(* IEC 61131-3 sources: SRCI/RobotLibrary/RobotLibrary/POUs/Calculation/MC_CalculateFrame, 1 file *)

(* ---- MC_CalculateFrameFB.st ---- *)
/// Calculate frame with three-point method
FUNCTION_BLOCK MC_CalculateFrameFB EXTENDS RobotLibraryBaseExecuteFB
// -------------------------------------------------------------------------
//  SRCI Robot Library
// -------------------------------------------------------------------------
//
//  Object:      CalculateFrameFB
//  Author:      Thorsten Brach
//  Date:        2024-06-09
//
//  Description:
//
//
//  Copyright:
//    (C) 2024 Thorsten Brach. All rights reserved
//             Licensed under the LGPL-3.0 license.
//
//  Disclaimer:
//    This project is provided without any guarantee and can be used for
//    private and commercial purposes. Any use is at the user’s
//    own risk and responsibility.
//
// -------------------------------------------------------------------------
VAR_INPUT
  /// command parameter
  ParCmd          : CalculateFrameParCmd;
END_VAR
VAR_OUTPUT
  /// Command is transferred and confirmed by the RC
  CommandBuffered : BOOL;
  /// Command output
  OutCmd          : CalculateFrameOutCmd;
END_VAR

VAR
  /// internal copy of command parameter
 _parCmd          : CalculateFrameParCmd;
  /// command data to send
 _command         : CalculateFrameSendData;
  /// response data received
 _response        : CalculateFrameRecvData;
  /// Incremented with each position of the input parameter "PositionsArray" sent from the PLC to the RC.
  /// Default: 0
 _dataIndex       : USINT;
  /// Set TRUE by the client, when according to the user selected "Mode" the final position of the input parameter "PositionsArray" is sent to the RC.
  /// Default: FALSE
 _dataComplete    : BOOL;
END_VAR

  SUPER^(AxesGroup := AxesGroup);

END_FUNCTION_BLOCK

METHOD CheckParameterChanged : BOOL
VAR_IN_OUT
  /// Robot assignment of function
  AxesGroup    : AxesGroup;
END_VAR

  // Check ParCmd Size is > 0, becaue MemCmp does not work correctly with size = 0
  IF (SIZEOF(ParCmd) = 0)
  THEN
    RETURN;
  END_IF

  // compare memory
  CheckParameterChanged := ( MemCmp(ADR(ParCmd), ADR(_parCmd), SIZEOF(ParCmd)) <> RobotLibraryConstants.OK );

  IF ( CheckParameterChanged )
  THEN
    // update internal copy of parameters
   _parCmd := ParCmd;
    // inc parameter sequence
   _command.ParSeq := _command.ParSeq + 1;
    // update command data
    CommandData := CreateCommandPayload(); // ( Access via reference to rCommandFB in ACR )
    // notify active command register
    AxesGroup.Acyclic.ActiveCommandRegister.NotifyParameterChanged := _uniqueID;
  END_IF

END_METHOD

METHOD INTERNAL CreateCommandPayload : SendData
// Table 6-656: Sent CMD payload (PLC to RC) of "CalculateFrame"
// --------------------------
// Header
// --------------------------
// Byte 00 : UINT       - Type HB
// Byte 01 :            - Type LB
// Byte 02 : USINT      - Reserve | ExecutionMode
// Byte 03 : USINT      - ParSeq  | Priority
// --------------------------
// Datablock
// --------------------------
// Byte 04 : USIN       - DataIndex
// Byte 05 : BOOL       - DataComplete
// Byte 06 : BYTE       - Reserve
// Byte 07 : USINT      - FrameNo
// Byte 08 : USINT      - ReferenceFrame
// Byte 09 : SINT       - Mode
// Byte 10 : REAL       - Position X  HW HB
// Byte 11 :            - Position X  HW LB
// Byte 12 :            - Position X  LW HB
// Byte 13 :            - Position X  LW LB
// Byte 14 : REAL       - Position Y  HW HB
// Byte 15 :            - Position Y  HW LB
// Byte 16 :            - Position Y  LW HB
// Byte 17 :            - Position Y  LW LB
// Byte 18 : REAL       - Position Z  HW HB
// Byte 19 :            - Position Z  HW LB
// Byte 20 :            - Position Z  LW HB
// Byte 21 :            - Position Z  LW LB
// Byte 22 : REAL       - Position Rx HW HB
// Byte 23 :            - Position Rx HW LB
// Byte 24 :            - Position Rx LW HB
// Byte 25 :            - Position Rx LW LB
// Byte 26 : REAL       - Position Ry HW HB
// Byte 27 :            - Position Ry HW LB
// Byte 28 :            - Position Ry LW HB
// Byte 29 :            - Position Ry LW LB
// Byte 30 : REAL       - Position Rz HW HB
// Byte 31 :            - Position Rz HW LB
// Byte 32 :            - Position Rz LW HB
// Byte 33 :            - Position Rz LW LB
// Byte 34 : Config     - ArmConfig   LW HB
// Byte 35 :            - ArmConfig   LW LB
// Byte 36 : TurnNumber - J1 + J2     LW HB
// Byte 37 :            - J3 + J4     LW LB
// Byte 38 :            - J5 + J6     LW LB
// Byte 39 :            - E1          LW LB
// Byte 40 : REAL       - Position E1 HW HB
// Byte 41 :            - Position E1 HW LB
// Byte 42 :            - Position E1 LW HB
// Byte 43 :            - Position E1 LW LB
// Byte 44 : REAL       - Position E2 HW HB
// Byte 45 :            - Position E2 HW LB
// Byte 46 :            - Position E2 LW HB
// Byte 47 :            - Position E2 LW LB
// Byte 48 : REAL       - Position E3 HW HB
// Byte 49 :            - Position E3 HW LB
// Byte 50 :            - Position E3 LW HB
// Byte 51 :            - Position E3 LW LB
// Byte 52 : REAL       - Position E4 HW HB
// Byte 53 :            - Position E4 HW LB
// Byte 54 :            - Position E4 LW HB
// Byte 55 :            - Position E4 LW LB
// Byte 56 : REAL       - Position E5 HW HB
// Byte 57 :            - Position E5 HW LB
// Byte 58 :            - Position E5 LW HB
// Byte 59 :            - Position E5 LW LB
// Byte 60 : REAL       - Position E6 HW HB
// Byte 61 :            - Position E6 HW LB
// Byte 62 :            - Position E6 LW HB
// Byte 63 :            - Position E6 LW LB
// --------------------------

  // set command parameter
  _command.CmdTyp         :=  CmdType.CalculateFrame;
  _command.ExecMode       :=  ExecMode;
  _command.ParSeq         := _command.ParSeq;
  _command.Priority       :=  Priority;
  _command.FrameNo        := _parCmd.FrameNo;
  _command.DataIndex      := _dataIndex;
  _command.DataComplete.0 := _dataComplete;
  _command.Reserve        := 0;
  _command.FrameNo        := _parCmd.FrameNo;
  _command.ReferenceFrame := _parCmd.ReferenceFrame;
  _command.Mode           := _parCmd.Mode;

  CASE _parCmd.Mode OF

    FrameCalculationMode.THREE_POINT_METHOD :

      CASE _dataIndex OF

        1: _command.Position := _parCmd.Origin;
        2: _command.Position := _parCmd.Position_X;
        3: _command.Position := _parCmd.Position_XY;

      END_CASE

    FrameCalculationMode.FOUR_POINT_METHOD  :

      CASE _dataIndex OF

        1: _command.Position := _parCmd.Origin;
        2: _command.Position := _parCmd.Position_X;
        3: _command.Position := _parCmd.Position_XY;
        4: _command.Position := _parCmd.OriginShift;

      END_CASE

    FrameCalculationMode.ONE_POINT_METHOD   :

     _command.Position := _parCmd.Origin;

  END_CASE

  // copy command data to header
  _cmdHeader := _command;
  // call base implementation to copy header to payload buffer
  CreateCommandPayload := SUPER^.CreateCommandPayload();

  // add command.DataIndex
  CreateCommandPayload.AddUsint(_command.DataIndex);
  // add command.DataComplete
  CreateCommandPayload.AddByte(_command.DataComplete);
  // add command.Reserve
  CreateCommandPayload.AddByte(_command.Reserve);
  // add command.FrameNo
  CreateCommandPayload.AddUsint(_command.FrameNo);
  // add command.ReferenceFrame
  CreateCommandPayload.AddUsint(_command.ReferenceFrame);
  // add command.Mode
  CreateCommandPayload.AddSint(_command.Mode);
  // add command.Position.X
  CreateCommandPayload.AddReal(_command.Position.X);
  // add command.Position.Y
  CreateCommandPayload.AddReal(_command.Position.Y);
  // add command.Position.Z
  CreateCommandPayload.AddReal(_command.Position.Z);
  // add command.Position.Rx
  CreateCommandPayload.AddReal(_command.Position.Rx);
  // add command.Position.Ry
  CreateCommandPayload.AddReal(_command.Position.Ry);
  // add command.Position.Rz
  CreateCommandPayload.AddReal(_command.Position.Rz);
  // add command.Position.Config
  CreateCommandPayload.AddArmConfig(_command.Position.Config);
  // add command.Position.TurnNumber
  CreateCommandPayload.AddTurnNumber(_command.Position.TurnNumber);
  // add command.Position.E1
  CreateCommandPayload.AddReal(_command.Position.E1);
  // add command.Position.E2
  CreateCommandPayload.AddReal(_command.Position.E2);
  // add command.Position.E3
  CreateCommandPayload.AddReal(_command.Position.E3);
  // add command.Position.E4
  CreateCommandPayload.AddReal(_command.Position.E4);
  // add command.Position.E5
  CreateCommandPayload.AddReal(_command.Position.E5);
  // add command.Position.E6
  CreateCommandPayload.AddReal(_command.Position.E6);

END_METHOD

METHOD FB_init : BOOL
VAR_INPUT
  /// if TRUE, the retain variables are initialized (warm start / cold start)
	bInitRetains : BOOL;
  /// if TRUE, the instance afterwards gets moved into the copy code (online change)
	bInCopyCode  : BOOL;
END_VAR

  MyType := 'MC_CalculateFrameFB';

  ExecMode := ExecutionMode.PARALLEL;

END_METHOD

METHOD PROTECTED OnCall
VAR_IN_OUT
  /// Robot assignment of function
  AxesGroup : AxesGroup;
END_VAR

  // call base implementation
  SUPER^.OnCall(AxesGroup := AxesGroup);

  CASE _stepCmd OF

    00:  IF ( _execute_R.Q )
         THEN
           // set busy flag
           Busy := TRUE;
           // Reset command outputs
           MemSet(ADR(OutCmd),0,SIZEOF(OutCmd));
           // apply command parameter
          _parCmd := ParCmd;
           // init parameter sequence
          _command.ParSeq := 1;
           // set timeout
           SetTimeout(PT := _timeoutCmd, rTimer := _timerCmd);
           // inc step counter
          _stepCmd := _stepCmd + 1;
  	     END_IF

    01: // inc data index
       _dataIndex := _dataIndex + 1;

        CASE _parCmd.Mode OF
          FrameCalculationMode.ONE_POINT_METHOD   :
            _dataComplete := _dataIndex >= 1;
          FrameCalculationMode.THREE_POINT_METHOD :
            _dataComplete := _dataIndex >= 3;
          FrameCalculationMode.FOUR_POINT_METHOD  :
            _dataComplete := _dataIndex >= 4;
  	    END_CASE

         // create command data
         CommandData := CreateCommandPayload();
         // Add command to active command register
        _uniqueID := AxesGroup.Acyclic.ActiveCommandRegister.AddCmd( pCommandFB := ADR(THIS^ ));
         // set timeout
         SetTimeout(PT := _timeoutCmd, rTimer := _timerCmd);
         // inc step counter
        _stepCmd := _stepCmd + 1;

    02:  // Wait for responce received
         IF ( _responseReceived )
         THEN
           // reset response received flag
          _responseReceived := FALSE;

           CASE  _response.State
           OF
             CmdMessageState.BUFFERED : CommandBuffered := TRUE;
             CmdMessageState.DONE     : Done            := TRUE;
             CmdMessageState.ERROR    : Error           := TRUE;
  				 END_CASE

           // Done, Aborted or Error ?
           IF (_response.State >= CmdMessageState.DONE )
           THEN
             // Reset Busy Flag
             Busy := FALSE;
             // Update results
             OutCmd.IEC_Date       := _response.IEC_Date;
             OutCmd.IEC_TIME       := _response.IEC_TIME;
             OutCmd.ReferenceFrame := _response.ReferenceFrame;
             OutCmd.Position       := _response.Position;

             IF ( _dataComplete ) OR (_response.State = CmdMessageState.ABORTED )
             THEN
               // set timeout
               SetTimeout(PT := _timeoutCmd, rTimer := _timerCmd);
               // inc step counter
              _stepCmd := _stepCmd + 1;
             ELSE
               // set timeout
               SetTimeout(PT := _timeoutCmd, rTimer := _timerCmd);
               // dec step counter
              _stepCmd := _stepCmd - 1;
  					 END_IF
  				 END_IF
         END_IF

    03: IF ( NOT Execute)
        THEN
          Reset();
  			END_IF
  ELSE
    // invalid step
    ErrorID := RobotLibraryEvents.ERR_INVALID_STEP;
  END_CASE

  // Cancel
  IF (Busy) AND (NOT Execute)
  THEN
    // try to remove cmd
    AxesGroup.Acyclic.ActiveCommandRegister.RemoveCmd(_uniqueID);
  END_IF

  // Reset FB
  IF ( NOT Execute )
  THEN
    Reset();
  END_IF

END_METHOD

METHOD INTERNAL ParseResponsePayload : DINT
// Table 6-657: Received CMD payload (RC to PLC) of "CalculateFrame"
// --------------------------
// Header
// --------------------------
// Byte 00 : USINT     - ParSeq | State
// Byte 01 : SINT      - AlarmMessageSeverity
// Byte 02 : UINT      - AlarmMessageCode HB
// Byte 03 :           - AlarmMessageCode LB
// --------------------------
// Datablock
// --------------------------
// Byte 04 : IEC_DATE  - FrameData.Date HB
// Byte 05 :           - FrameData.Date LB
// Byte 06 : IEC_TIME  - FrameData.Time HB HW
// Byte 07 :           - FrameData.Time HB LW
// Byte 08 :           - FrameData.Time LW HB
// Byte 09 :           - FrameData.Time LW LB
// Byte 10 : USINT     - FrameData.ReferenceFrame
// Byte 11 : BYTE      - Reserve
// Byte 12 : REAL      - FrameData.X  HB HW
// Byte 13 :           - FrameData.X  HB LW
// Byte 14 :           - FrameData.X  LW HB
// Byte 15 :           - FrameData.X  LW LB
// Byte 16 : REAL      - FrameData.Y  HB HW
// Byte 17 :           - FrameData.Y  HB LW
// Byte 18 :           - FrameData.Y  LW HB
// Byte 19 :           - FrameData.Y  LW LB
// Byte 20 : REAL      - FrameData.Z  HB HW
// Byte 21 :           - FrameData.Z  HB LW
// Byte 22 :           - FrameData.Z  LW HB
// Byte 23 :           - FrameData.Z  LW LB
// Byte 24 : REAL      - FrameData.Rx HB HW
// Byte 25 :           - FrameData.Rx HB LW
// Byte 26 :           - FrameData.Rx LW HB
// Byte 27 :           - FrameData.Rx LW LB
// Byte 28 : REAL      - FrameData.Ry HB HW
// Byte 29 :           - FrameData.Ry HB LW
// Byte 30 :           - FrameData.Ry LW HB
// Byte 31 :           - FrameData.Ry LW LB
// Byte 32 : REAL      - FrameData.Rz HB HW
// Byte 33 :           - FrameData.Rz HB LW
// Byte 34 :           - FrameData.Rz LW HB
// Byte 35 :           - FrameData.Rz LW LB
// --------------------------
VAR_INPUT
  /// Response data
  ResponseData : RecvData;
END_VAR

  // call base implementation to parse the header from payload buffer
  ResponseData.PayloadPtr := SUPER^.ParseResponsePayload(ResponseData);

  // copy parsed header to response
  _response.ParSeq               := _rspHeader.ParSeq;
  _response.State                := _rspHeader.State;
  _response.AlarmMessageSeverity := _rspHeader.AlarmMessageSeverity;
  _response.AlarmMessageCode     := _rspHeader.AlarmMessageCode;

  // Get response.IEC_Date
  _response.IEC_Date   := ResponseData.GetIecDate();
  // Get response.IEC_TIME
  _response.IEC_TIME   := ResponseData.GetIecTime();
  // Get response.ReferenceFrame
  _response.ReferenceFrame := ResponseData.GetUsint();
  // Get response.Reserve
  _response.Reserve := ResponseData.GetByte();
  // Get response.Position.X
  _response.Position.X := ResponseData.GetReal();
  // Get response.Position.Y
  _response.Position.Y := ResponseData.GetReal();
  // Get response.Position.Z
  _response.Position.Z := ResponseData.GetReal();
  // Get response.Position.Rx
  _response.Position.Rx := ResponseData.GetReal();
  // Get response.Position.Ry
  _response.Position.Ry := ResponseData.GetReal();
  // Get response.Position.Rz
  _response.Position.Rz := ResponseData.GetReal();

END_METHOD

METHOD PROTECTED Reset : DINT
VAR_INPUT
END_VAR

  Reset := SUPER^.Reset();

  Done               := FALSE;
  Busy               := FALSE;
  CommandBuffered    := FALSE;

END_METHOD
